// TIA Portal V20 export
TYPE "UDT_AnaSlot"
// AI/AQ module slot 4-20mA
   STRUCT
      Enable : Bool;
      StartAddr : UInt;
      ChannelCount : USInt;
      Reserved : USInt;
      RawFull : Int := 27648;
      EngMax_mA : Real := 20.0;
      EngMin_mA : Real := 4.0;
   END_STRUCT;
END_TYPE
